// TIA Portal V19 export
TYPE "Time Zone"
   STRUCT
      City : String;
      "Local Time" : Time_Of_Day;
      Offset : Time;
   END_STRUCT;
END_TYPE
